TYPE INTERNAL ST_Entry :
STRUCT
	iSignal		: I_SignalNode;
	iReceiver	: I_ReceiverNode;
END_STRUCT
END_TYPE

(* stored: Version 1.1.0.1
   DUT ST_Entry: Id {bdd102f7-97bb-4876-8491-edc279268ab7} *)
